PROGRAM P_GeneralStateManager
VAR
	(*
		Author - Gideon Jgordon (GJ)
		Changes 
		-(GJ) Added to govern the General State of the STS04 Machine 
		-(GJ) stGSM moved to P_AllStateChecker to make it cleaner
	*)	
	nStateGeneral : INT;
	bValuesResetDone: BOOL;
END_VAR

CASE nStateGeneral OF

GeneralStateMain.State_Init				: //Initialize all the state

	IF gvl.stHMI.bStart THEN
		nStateGeneral:= GeneralStateMain.State_Reset;
		ELSE
		nStateGeneral:=	GeneralStateMain.State_Init;
	END_IF	
	
GeneralStateMain.State_Reset			: // Reset behaviour and values befor we proceed to go into Run Mode

	//Adding reset below here
	IF (bValuesResetDone AND P_AllStateChecker.bAllOk) THEN
		nStateGeneral:=GeneralStateMain.State_Run;
		gvl.stGSM.bStart	:=TRUE;
	END_IF
	IF NOT (bValuesResetDone AND P_AllStateChecker.bAllOk) THEN
		nStateGeneral:=GeneralStateMain.State_Init;
	END_IF
	
GeneralStateMain.State_Run              : // Governs the Process during run

	IF NOT P_AllStateChecker.bAllOk THEN
		gvl.stGSM.bStart	:=FALSE;
	END_IF
	IF gvl.stHMI.bStop THEN
		nStateGeneral:= GeneralStateMain.State_Stop;
		gvl.stGSM.bStart	:=FALSE;
	END_IF
	
GeneralStateMain.State_Stop             : //Stop via HMI or Error

	nStateGeneral:= GeneralStateMain.State_Init;
	
GeneralStateMain.State_ErrorCheck       :

	
	
END_CASE

END_PROGRAM

(* stored: Version 1.1.0.1, ProductVersion 3.1.4024.12
   POU P_GeneralStateManager: Id {527686d1-db88-4d1f-8d7e-14a8310b3953}, SpecialFunc None *)
